PROGRAM MAIN
VAR
	Galaxy : Galaxy;
END_VAR

// Init - First Scan Done before run Galaxy
IF NOT Galaxy.IsInitialized THEN
	Galaxy.Init();
	RETURN;
END_IF

// Cyclic
Galaxy();

END_PROGRAM

(* stored: Version 1.1.0.1
   POU MAIN: Id {f9ecec64-8aac-48a0-8b4b-5617ed442c3a}, SpecialFunc None *)
